FUNCTION_BLOCK FB_LogHandler_PersistentArray EXTENDS FB_LogHandlerBase // Writes the last X-number of log items to a persistent list
VAR PERSISTENT
	aLogItems : ARRAY[1..GVL_Utilities.RETAINABLE_LOG_HISTORY_SIZE] OF UDT_LogItem;
	nIndex : UINT; // Array index of the last added log item
END_VAR
VAR
	nIterIndex : UINT; // Array index of the iterator
END_VAR

METHOD INTERNAL FINAL AddToLog
VAR_INPUT
	stLogItem : UDT_LogItem;
END_VAR
VAR
	i : UINT; // Iterator
END_VAR
nIndex := (nIndex MOD GVL_Utilities.RETAINABLE_LOG_HISTORY_SIZE) + 1;
aLogItems[nIndex] := stLogItem;
END_METHOD

METHOD PROTECTED Get : UDT_LogItem // Get logitem based on nIterIndex; return an empty logitem if index is invalid
VAR
	stEmptyLogItem : UDT_LogItem;
END_VAR
IF (nIterIndex >= 1) AND (nIterIndex <= GVL_Utilities.RETAINABLE_LOG_HISTORY_SIZE) THEN
	Get := aLogItems[nIterIndex];
ELSE
	Get := stEmptyLogItem;
END_IF
END_METHOD

METHOD PUBLIC Last : UDT_LogItem // Return the last added logitem
nIterIndex := nIndex;
Last := Get();
END_METHOD

METHOD PUBLIC Previous : UDT_LogItem // Return the logitem previous to the one got before using Last() or Previous()
nIterIndex := nIterIndex - 1;
IF (nIterIndex = 0) THEN // Roll over when lower bound is reached
	nIterIndex := GVL_Utilities.RETAINABLE_LOG_HISTORY_SIZE;
END_IF
Previous := Get();
END_METHOD

END_FUNCTION_BLOCK

(* stored: Version 1.1.0.1, ProductVersion 3.1.4024.11
   POU FB_LogHandler_PersistentArray: Id {4966cdb4-950f-0659-2a45-e07380f91fca}, SpecialFunc None
   Method AddToLog: Id {10aa411e-05f8-09bd-04b5-bb2a775a1d6a}
   Method Get: Id {b92d4215-1114-0c08-3493-8db7b8a0c244}
   Method Last: Id {96b46594-086e-0228-303b-2e866d241c47}
   Method Previous: Id {2b4efa5f-2fea-0055-281f-6f818d469f92} *)
